{attribute 'qualified_only'}
{attribute 'strict'}
{attribute 'to_string'}
TYPE OpState :
(
	OP 		:= 0,
	NOT_OP	:= 1
) DINT;
END_TYPE

(* stored: Version 1.1.0.1, ProductVersion 3.1.4026.6
   DUT OpState: Id {6332afc8-51f0-477e-817f-8f663c228f05} *)
